// TIA Portal V15.1 export
// export: Created 2020-12-23T11:47:33.918068Z, ExportSetting WithDefaults, WithReadOnly, DisplayName Totally Integrated Automation Portal, DisplayVersion V15.1 Update 3, DisplayName TIA Portal Openness, DisplayVersion V15.1, DisplayName STEP 7 Professional, DisplayVersion V15.1 Update 3, DisplayName WinCC Advanced, DisplayVersion V15.1 Update 3
VAR_GLOBAL   // PLC tag table "io_import"
END_VAR
